PROGRAM MAIN
VAR
		Burner_1 :Burner_Main;
END_VAR

Burner_1();

END_PROGRAM

(* stored: Version 1.1.0.1
   POU MAIN: Id {cf356ef4-b289-4228-a8ea-3f3b2b219387}, SpecialFunc None *)
